TYPE ST_InputsSubsystemManager :
(**************************************************************************************
 * 	Application		:	BoxControl Framework
 *	Revision		:	$Revision: 404529 $
 *	Revision date	:	$Date: 2018-04-23 08:21:38 +0200 (Mo., 23 Apr 2018) $
 *	Last changed by	:	$Author: b7bolm $
 *	URL				:	$URL: http://almscdc.swisslog.com/repo/SWPD/Development/BoxControlFramework/20_Release/trunk/01_Software/BCF/BCF/JumpStart/20_Product/10_App/15_Subsystem/10_Lib/10_Conv/01_DUTs/10_Dummy/ST_InputsSubSystemManager.TcDUT $
 *
 *	Purpose			:	Inputs Subsystem manager
 *
 * ------------------------------------------------------------------------------------
 *	Copyright Swisslog [IP AG], Switzerland. All rights reserved.
 * 
 * ------------------------------------------------------------------------------------
 *	
 * 	Revision History: 
 *
 * 	VERSION			DATE			INITIALS			DESCRIPTION
 *	0.1				01.01.2001		swl					Example
 *
 **************************************************************************************)
STRUCT
	EtherCAT_MasterState			: UINT; // Diagnostic info of EtherCat Master node 
	EtherCAT_MasterWorkingCounter	: UINT; // Diagnostic info of EtherCat Master node 
	FanSpeed						: UINT; // Fan speed
	CPU_Temperatur					: INT; // Temp CPU  
	CPU_Usage						: INT; // Usage CPU
	SystemUsage						: INT; // Usage System
	DeviceState	  					: ARRAY [1..400] OF UINT; // Diagnostic info of EtherCAT slave devices
END_STRUCT
END_TYPE

(* stored: Version 1.1.0.1, ProductVersion 3.1.4022.12
   DUT ST_InputsSubSystemManager: Id {85284f7e-77b9-4a4e-bf91-a00b0cc04b8c} *)
